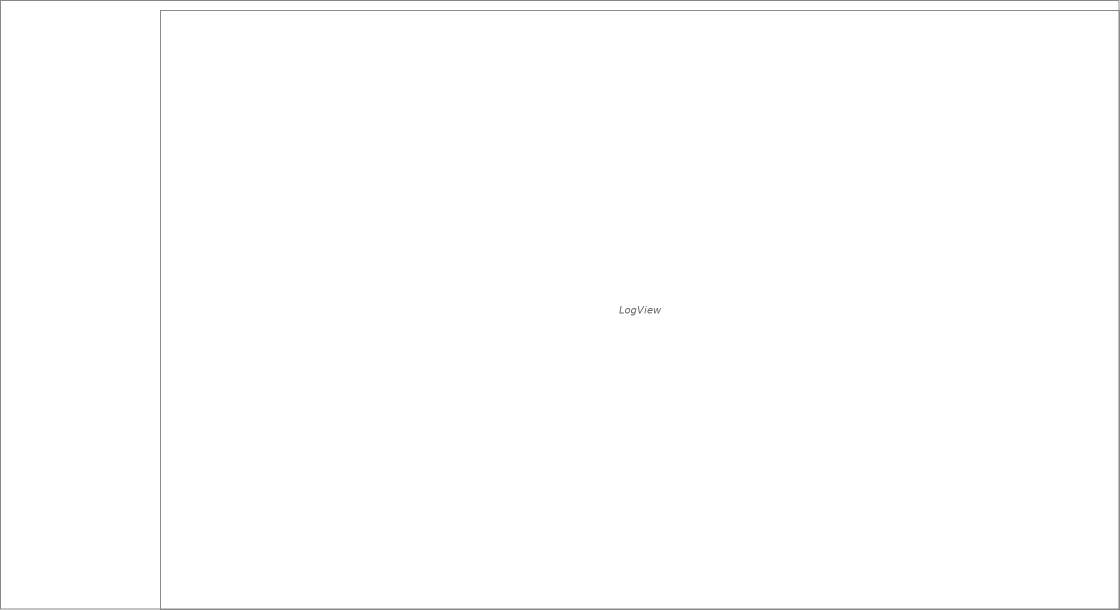
VISUALIZATION FaultLog  // 1120x610
VAR_IN_OUT
	fbLogger : FB_Logger;
END_VAR
    Frame (160,10 960x600)
        shows LogView(fbLogView := GVL_HMI.fbHMIControl.fbLogView)
        [0]: fbLogger=fbLogger
END_VISUALIZATION

(* stored: Version 1.1.0.1, ProductVersion 3.1.4024.11
   Visu FaultLog: Id {9d1d492b-4ead-40bc-8482-c9349fd92015} *)
